FUNCTION_BLOCK DoorModel (* Composite Function Block Type *)
  (* Standard: 61499-2 *)
  (* Version 1.0, 2019-05-07, jetbrains *)
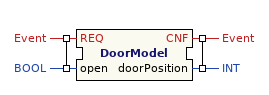
  EVENT_INPUT
    REQ WITH open; (* Normal Execution Request *)
  END_EVENT
  EVENT_OUTPUT
    CNF WITH doorPosition; (* Execution Confirmation *)
  END_EVENT
  VAR_INPUT
    open : BOOL; (* Input event qualifier *)
  END_VAR
  VAR_OUTPUT
    doorPosition : INT; (* Output event qualifier *)
  END_VAR
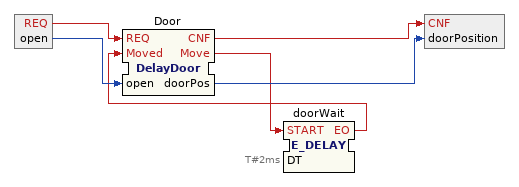
  FBS
    doorWait : E_DELAY(DT := T#2ms);
    Door : DelayDoor;
  END_FBS
  EVENT_CONNECTIONS
    REQ TO Door.REQ;
    doorWait.EO TO Door.Moved;
    Door.CNF TO CNF;
    Door.Move TO doorWait.START;
  END_CONNECTIONS
  DATA_CONNECTIONS
    open TO Door.open;
    Door.doorPos TO doorPosition;
  END_CONNECTIONS
END_FUNCTION_BLOCK
